// This function has been automatically generated from the project information.
{attribute 'signature_flag' := '1073741824'}
{attribute 'TcGenerated'}
{attribute 'no-analysis'}
FUNCTION F_GetTitle : WSTRING
VAR_INPUT
	
END_VAR

F_GetTitle := "Workshop Library";

END_FUNCTION

(* stored: Version 1.1.0.1
   POU F_GetTitle: Id {3562fab7-6986-480d-a78b-9143225be5cb}, SpecialFunc None *)
